FUNCTION_BLOCK ValveS (* CAT Function Block Type *)
  (* Standard: 61499-2 *)
  (* Version 0.0, 6/2/2026, Schneider Electric, template *)
  PACKAGE SE.Nereda;
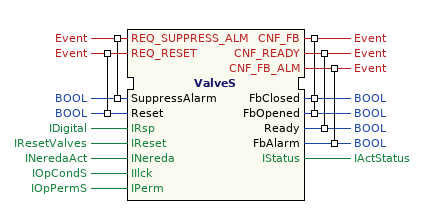
  EVENT_INPUT
    REQ_SUPPRESS_ALM WITH SuppressAlarm; (* Request to update the alarm suppress status *)
    REQ_RESET WITH Reset; (* Request to reset the device *)
  END_EVENT
  EVENT_OUTPUT
    CNF_FB WITH FbClosed, FbOpened; (* Execution of confirmed state *)
    CNF_READY WITH Ready; (* Execution of Ready status *)
    CNF_FB_ALM WITH FbAlarm; (* Execution of confirmation  Fb alarm *)
  END_EVENT
  VAR_INPUT
    SuppressAlarm : BOOL; (* 1 = Suppress alarm in HMI *)
    Reset : BOOL; (* 1 = Reset device failure *)
  END_VAR
  VAR_OUTPUT
    FbClosed : BOOL; (* 1 = Stopped *)
    FbOpened : BOOL; (* 1 = Running *)
    Ready : BOOL; (* 1 = Device is ready to run *)
    FbAlarm : BOOL; (* 1 = Feedback failure alarm is active *)
  END_VAR
  SOCKETS
    IRsp : IDigital;
    IReset : IResetValves;
    INereda : INeredaAct(pin_6EEAF63EEE6021B6 := FALSE);
  END_SOCKETS
  SOCKETS
    IIlck : IOpCondS; (* Condition summary chain input from upstream blocks *)
    IPerm : IOpPermS; (* Permission condition summary chain input from permCondItem blocks *)
  END_SOCKETS
  PLUGS
    IStatus : IActStatus;
  END_PLUGS
  (* 01 - FUNCTIONNAL INPUT INTERFACE *)
  (* 00 - INITIALIZATION *)
  (* 05 - LOGIC *)
  (* 06 - HMI INTERFACE *)
  (* 04 - CHILDREN *)
  (* 03 - FIELD INTERFACE *)
  (* 02 - FUNCTIONNAL OUTPUT INTERFACE *)
  (* 07- Input Hardware Interface *)
  (* 08- Output Hardware Interface *)
  (* 09- Local Panel *)
  (* Maintenance *)
  (* Cmd Out *)
  (* Interlock *)
  (* Mode *)
  (* Permissive *)
  (* 4A - TYPICALS *)
  (* Reset *)
  (* Cmd *)
  (* Simulation (To be Removed) *)
  FBS
    IThis : ValveS_HMI(QI := TRUE);
    INIT : plcStart(Prio := 35, Delay := T#0ms);
    extControlled : dISignal(Name := '$${PATH}DIn'); {SET_ATTRIBUTE(Configuration.Component.HideUnusedPorts, )}
    cmdOpen : dOSignal(Name := '$${PATH}DOut'); {SET_ATTRIBUTE(Configuration.Component.HideUnusedPorts, )}
    LocalPanel : FieldSignals;
    maintenance : DevMnt(StateSel := Motor); {SET_ATTRIBUTE(Configuration.Component.HideUnusedPorts, )}
    interlock : IlckCondSum; {SET_ATTRIBUTE(Configuration.Component.HideUnusedPorts, )}
    CurrOwner : CurrOwnerDecode;
    State : ActState(pin_DD241BABAE81E6FD := Valve, pin_94E3C396E1CCD1C0 := FALSE, pin_C70237F918BB93F6 := TRUE);
    permissive : PermCondSum; {SET_ATTRIBUTE(Configuration.Component.HideUnusedPorts, )}
    ResetCmd : OR_169B00D031196E7C4; {SET_ATTRIBUTE(Configuration.GenericFBType.InterfaceParams, Runtime.Standard#CNT:=4;OUT:BOOL)}
    Base : ValveBase;
    fbOpen : dISignal(Name := '$${PATH}DIn'); {SET_ATTRIBUTE(Configuration.Component.HideUnusedPorts, )}
    fbClose : dISignal(Name := '$${PATH}DIn'); {SET_ATTRIBUTE(Configuration.Component.HideUnusedPorts, )}
    CmdOut : CmdDecode;
    cmdClose : dOSignal(Name := '$${PATH}DOut'); {SET_ATTRIBUTE(Configuration.Component.HideUnusedPorts, )}
    IRspDecode : ValveSpDecode;
    Sp : DS_SELECTX_6147A5438F26867; {SET_ATTRIBUTE(Configuration.GenericFBType.InterfaceParams, Runtime.Standard#CNTX:=2;CNTY:=1;DI${CNTX,_,CNTY$}:INT)}
    cmdopenname : VALFORMAT_1798710A2657A9EEF(VALUE1 := '$${PATH:0,0}', FORMAT := '%s.%s', VALUE2 := 'cmdOpen.DOut'); {SET_ATTRIBUTE(Configuration.GenericFBType.InterfaceParams, Runtime.Standard#I:=2;VALUE${I$}:STRING,STRING)}
    fbopenname : VALFORMAT_1798710A2657A9EEF(VALUE1 := '$${PATH:0,0}', FORMAT := '%s.%s', VALUE2 := 'fbOpen.DIn'); {SET_ATTRIBUTE(Configuration.GenericFBType.InterfaceParams, Runtime.Standard#I:=2;VALUE${I$}:STRING,STRING)}
    fbpowername : VALFORMAT_1798710A2657A9EEF(VALUE1 := '$${PATH:0,0}', FORMAT := '%s.%s', VALUE2 := 'LocalPanel.PowerFb'); {SET_ATTRIBUTE(Configuration.GenericFBType.InterfaceParams, Runtime.Standard#I:=2;VALUE${I$}:STRING,STRING)}
    fbatvrdyname : VALFORMAT_1798710A2657A9EEF(VALUE1 := '$${PATH:0,0}', FORMAT := '%s.%s', VALUE2 := 'LocalPanel.AtvReady'); {SET_ATTRIBUTE(Configuration.GenericFBType.InterfaceParams, Runtime.Standard#I:=2;VALUE${I$}:STRING,STRING)}
    cmdclosename : VALFORMAT_1798710A2657A9EEF(VALUE1 := '$${PATH:0,0}', FORMAT := '%s.%s', VALUE2 := 'cmdClose.DOut'); {SET_ATTRIBUTE(Configuration.GenericFBType.InterfaceParams, Runtime.Standard#I:=2;VALUE${I$}:STRING,STRING)}
    fbclosename : VALFORMAT_1798710A2657A9EEF(VALUE1 := '$${PATH:0,0}', FORMAT := '%s.%s', VALUE2 := 'fbClose.DIn'); {SET_ATTRIBUTE(Configuration.GenericFBType.InterfaceParams, Runtime.Standard#I:=2;VALUE${I$}:STRING,STRING)}
    Sim : ActuatorsSimulation;
    TriggerCmd : RetriggerEvent(pin_CFF51EFF0A91DC53 := 3, pin_FDD5DC24A8674AF6 := T#1s);
  END_FBS
  EVENT_CONNECTIONS
    extControlled.CNF TO Base.REQ_EXT_CTL;
    fbClose.CNF TO Base.REQ_FB;
    interlock.COND_IND TO Base.REQ_ILCK;
    REQ_SUPPRESS_ALM TO Base.REQ_SUPPRESS_ALM;
    Base.CNF_FB_STS TO CNF_FB;
    Base.CNF_FB_ALM TO CNF_FB_ALM;
    Base.CNF_OUT TO maintenance.REQ;
    Base.CNF_FB_ALM TO maintenance.REQ_ALM;
    Base.CNF_MODE TO maintenance.REQ;
    REQ_SUPPRESS_ALM TO maintenance.REQ_SUPPRESS_ALM;
    permissive.PERM_IND TO Base.REQ_PERM;
    IRsp.REQ TO Sp.REQ1;
    REQ_RESET TO ResetCmd.REQ;
    ResetCmd.CNF TO Base.REQ_RESET;
    fbpowername.CNF TO fbatvrdyname.REQ;
    cmdopenname.CNF TO cmdclosename.REQ;
    fbopenname.CNF TO fbclosename.REQ;
    cmdclosename.CNF TO fbopenname.REQ;
    fbclosename.CNF TO fbpowername.REQ;
    fbOpen.CNF TO Base.REQ_FB;
    LocalPanel.08EBB16DA2AE2E53 TO CurrOwner.3D8B91432EBB5812;
    IReset.DB2F31576D7C8341 TO ResetCmd.REQ;
    Base.CNF_NEED_RESET TO IReset.6762F1A42616FBAF;
    Base.CNF_FB_STS TO INereda.9CD053F8408797ED;
    State.3E2F994B40CA5D8A TO INereda.CC753684FA882790;
    Base.CNF_FB_ALM TO INereda.C79FD2A34D0395C5;
    maintenance.CNF_OPD TO INereda.2DA8AEC15204E92D;
    INereda.0F1CDF9A9B4A227A TO Sp.REQ2;
    INereda.37BBC1F841739733 TO ResetCmd.REQ;
    CurrOwner.7B1DE71047870DF3 TO State.503DFB34A9D9F842;
    State.B9B326A02DDC85D5 TO INIT.ACK_FIRST;
    State.B9B326A02DDC85D5 TO cmdopenname.REQ;
    Sp.IND TO IRspDecode.6ADB36776E847893;
    TriggerCmd.4002AEF0814D09CF TO Base.REQ_SP;
    Base.CNF_OUT TO CmdOut.A84FFA5C79DEC05E;
    CmdOut.7DBA80A4DCA36C5D TO cmdOpen.REQ;
    CmdOut.7DBA80A4DCA36C5D TO cmdClose.REQ;
    State.3E2F994B40CA5D8A TO CNF_READY;
    Base.CNF_FB_STS TO IStatus.14377629A1F197A9;
    State.3E2F994B40CA5D8A TO IStatus.14377629A1F197A9;
    Base.CNF_SP TO CurrOwner.3D8B91432EBB5812;
    Base.CNF_FB_STS TO CurrOwner.3D8B91432EBB5812;
    Base.CNF_READY TO CurrOwner.3D8B91432EBB5812;
    Base.CNF_OWNER TO CurrOwner.3D8B91432EBB5812;
    Base.CNF_MODE TO CurrOwner.3D8B91432EBB5812;
    interlock.COND_IND TO CurrOwner.3D8B91432EBB5812;
    IRspDecode.9274835450AA07E7 TO TriggerCmd.2BC1963D96179493;
    Base.CNF_OWNER TO IRspDecode.6ADB36776E847893;
    Base.CNF_FB_ALM TO CurrOwner.3D8B91432EBB5812;
    Base.CNF_NEED_RESET TO CurrOwner.3D8B91432EBB5812;
    fbatvrdyname.CNF TO Sim.1F0D1F6D665FD1A3;
    INIT.REDO_INIT TO IThis.5D65C7F23F6CCFDB;
    INIT.FIRST_INIT TO IThis.5D65C7F23F6CCFDB;
    State.B9B326A02DDC85D5 TO IThis.D29F1FADF6E57358;
    Base.CNF_NEED_RESET TO IThis.56CAC1A52910316B;
    maintenance.CNF_OPD TO IThis.DB5D3D5EB4CA50A8;
    State.7E9F7DF9BBDC513D TO IThis.115F74063274DE8D;
    fbClose.CNF TO IThis.9B561975ECC81360;
    fbOpen.CNF TO IThis.9B561975ECC81360;
    IThis.141F2765F0199247 TO State.747A80A26976E9BA;
    IThis.A591CDF920E284FE TO ResetCmd.REQ;
  END_CONNECTIONS
  DATA_CONNECTIONS
    extControlled.Out TO Base.ExternalControlled;
    fbOpen.Out TO Base.FbOpen;
    fbClose.Out TO Base.FbClose;
    interlock.CondPos TO Base.IlckPos;
    interlock.CondType TO Base.IlckType;
    interlock.State TO Base.IlckCond;
    SuppressAlarm TO Base.SuppressAlarm;
    Base.FbClosed TO FbClosed;
    Base.FbOpened TO FbOpened;
    Base.FbAlarm TO FbAlarm;
    Base.Out TO maintenance.Pv;
    Base.FbAlarm TO maintenance.DeviceAlarm;
    Base.Simulation TO maintenance.Sim;
    SuppressAlarm TO maintenance.SuppressAlarm;
    permissive.PermPassive TO Base.PermClose;
    permissive.PermActive1 TO Base.PermOpen;
    IRsp.Value TO Sp.DI1_1;
    Reset TO ResetCmd.IN1;
    ResetCmd.OUT TO Base.Reset;
    LocalPanel.B46B24B64003C584 TO State.655DE7D6E2CF8FB8;
    IReset.C45940A1007F76EB TO ResetCmd.IN3;
    Base.NeedReset TO IReset.175754047DFBD268;
    Base.FbOpened TO INereda.7F6CC7FEB9223DF3;
    Base.FbClosed TO INereda.A8D6C4A1FDCCA991;
    State.4E509FA35DBACB85 TO INereda.8A8A07EFCDA1443C;
    Base.FbAlarm TO INereda.BDD69968F2D82EAF;
    maintenance.TotalOperationDuration TO INereda.C7F638DBF6B860D2;
    maintenance.CurrentOperationDuration TO INereda.9224E22E0E82A2D7;
    maintenance.OperationCount TO INereda.10624535249F94F3;
    INereda.710D7FC54EE3F35A TO Sp.DI2_1;
    INereda.EA28053F07575F36 TO ResetCmd.IN4;
    CurrOwner.CEBE936F1EA616DB TO State.E90E39DE4A80ABDE;
    CurrOwner.1FF13EB8D921FC26 TO State.3885B231A80F7FFF;
    Base.CurrentSp TO State.52C3EF6D9E750127;
    Base.FbStatus TO State.8E076A9FED13120E;
    Base.Ready TO State.1C9201C719ABF50B;
    Base.Simulation TO State.7A0BDA68B634A263;
    Base.FbOverride TO State.DD66F5DCF7F6FB1D;
    interlock.State TO State.9A204E382C1350DC;
    Sp.OUT1 TO IRspDecode.E3DBDFEF31CE8CF0;
    IRspDecode.2CEC9083D9D2002C TO Base.Sp;
    Base.Out TO CmdOut.AB3CA6CBC1A8076E;
    CmdOut.3DD5E33A07331CE4 TO cmdOpen.Signal;
    CmdOut.098895859CE66202 TO cmdClose.Signal;
    State.4E509FA35DBACB85 TO Ready;
    Base.FbOpened TO IStatus.72E790857420193D;
    Base.FbClosed TO IStatus.3A653A8838D163CA;
    State.4E509FA35DBACB85 TO IStatus.9E0B44559326BEAF;
    Base.CurrentOwner TO CurrOwner.B2DAC483AB345195;
    cmdopenname.RESULT TO Sim.CF35C6FFF71E6DA9;
    cmdclosename.RESULT TO Sim.A062E8F5348A5B29;
    fbopenname.RESULT TO Sim.DA56AF0AB63864EC;
    fbclosename.RESULT TO Sim.8527B15BE9544648;
    fbpowername.RESULT TO Sim.B9574325CA25CB90;
    fbatvrdyname.RESULT TO Sim.BC3DC36B550BA99C;
    Base.FbAlarm TO State.F37ACDE435F84908;
    Base.NeedReset TO State.3ED730632EF45559;
    Base.NeedReset TO IThis.40C9F9C762B4EBFC;
    maintenance.CurrentOperationDuration TO IThis.F72B4FFB993E14D8;
    State.8CCAFBE354ECA569 TO IThis.A4F116D0A19D9B8F;
    fbClose.Out TO IThis.1F7B63A485BAF943;
    IThis.E6FBA099621F55FB TO ResetCmd.IN2;
    fbOpen.Out TO IThis.F1FF7ECA794BAF00;
  END_CONNECTIONS
  ADAPTER_CONNECTIONS
    IIlck TO interlock.IOpCondIn;
    IPerm TO permissive.IOpPermIn;
  END_CONNECTIONS
END_FUNCTION_BLOCK
